VISUALIZATION VISU_DEBUG  // 2x2
END_VISUALIZATION

(* stored: Version 1.1.0.1, ProductVersion 3.1.4024.0
   Visu VISU_DEBUG: Id {ab3ba7f3-f971-4ccd-b938-5f04d7f3ff01} *)
